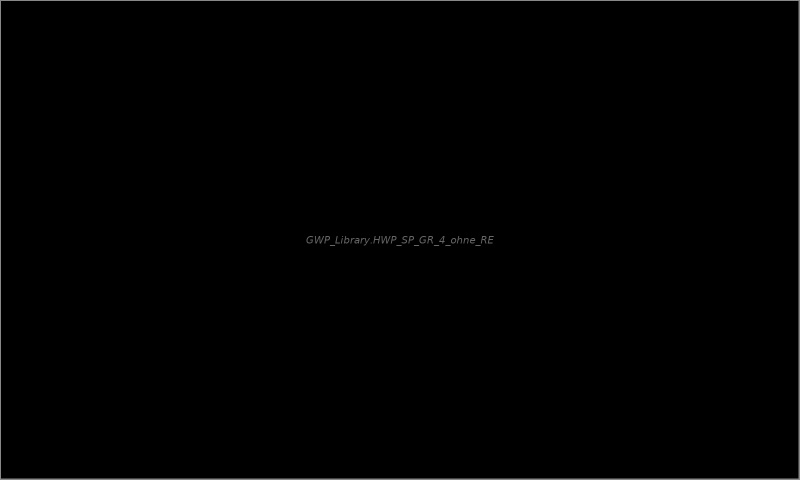
VISUALIZATION HWP_SP_GR_4_ohne_RE  // 800x480
    Frame (0,0 800x480)
        shows GWP_Library.HWP_SP_GR_4_ohne_RE(FB_GR_4_ohne_RE := Main.HWP_SP_0.GR_4_ohne_RE_0, FB_Init_1 := Main.Init_0)
END_VISUALIZATION

(* stored: Version 1.1.0.1, ProductVersion 3.1.4022.6
   Visu HWP_SP_GR_4_ohne_RE: Id {6c0c3754-c2b8-4c63-8a2a-367b391b61df} *)
